TYPE E_DataExchaSteps :
(
	DATAEXCHA_STATE_IDLE,
	DATAEXCHA_STATE_SEND_START,
	DATAEXCHA_STATE_SEND_WAIT,
	DATAEXCHA_STATE_RECEIVE_START,
	DATAEXCHA_STATE_RECEIVE_WAIT,
	DATAEXCHA_STATE_ERROR
);
END_TYPE

(* stored: Version 1.1.0.1, ProductVersion 3.1.4024.12
   DUT E_DataExchaSteps: Id {0624b23b-52ee-4031-ad25-f12c5a71eb72} *)
